// TIA Portal V20 export
FUNCTION "FC_ExtractGripper" : Void   // FC9, LAD
{ S7_Optimized_Access := 'TRUE' }
// stored: SetENOAutomatically false
   VAR_INPUT
      GripperVal : DInt;
   END_VAR
   VAR_OUTPUT
      Gripper1 : Int;
      Gripper2 : Int;
   END_VAR
BEGIN

REGION Network 1 (SCL)
   IF #GripperVal < 1000 THEN
       #Gripper1 := DINT_TO_INT(#GripperVal);
       #Gripper2 := 0;
   ELSE
       #Gripper1 := TRUNC_INT(#GripperVal / 1000);
       #Gripper2 := DINT_TO_INT(#GripperVal ) - (TRUNC_INT(#GripperVal / 1000) * 1000);
   END_IF;
END_REGION
END_FUNCTION
